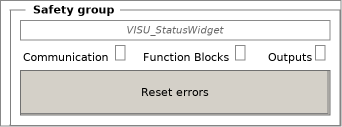
VISUALIZATION VISU_SafetyGroup  // 342x127
VAR_IN_OUT
    statusWidget : StatusWidget;
    comError : BOOL;
    fbError : BOOL;
    outError : BOOL;
    reset : Process;
END_VAR
    Polyline (25,10) (10,10) (10,125) (340,125) (340,10) (120,10)
    Label (30,0 125x20), "Safety group"
    Label (20,45 90x25), "Communication"
    Label (140,45 90x25), "Function Blocks"
    Label (265,45 55x25), "Outputs"
    Frame (115,45 10x15)
        shows VISU_State_green_red(state := comError)
    Frame (235,45 10x15)
        shows VISU_State_green_red(state := fbError)
    Frame (315,45 10x15)
        shows VISU_State_green_red(state := outError)
    Frame (20,20 310x20)
        shows VISU_StatusWidget(widget := statusWidget)
    Button (20,70 310x45), "Reset errors", input disabled if: reset.statuses.enabledStatus.disabled
        OnMouseClick: execute { reset.do_request := TRUE; }
END_VISUALIZATION

(* stored: Version 1.1.0.1, ProductVersion 3.1.4019.2
   Visu VISU_SafetyGroup: Id {40be5b69-0377-4b46-bea6-3b784f5f7bf0} *)
